FUNCTION FB_HEXSTR_TO_DINT																			// Converts a STRING hex array to DINT.
VAR_INPUT
	in						: STRING;																// The input string.
END_VAR
VAR_OUTPUT
	out						: DINT;																	// The output value.
	bError					: BOOL;																	// Had any error occured.
END_VAR
VAR
	sSum					: STRING;
	pVal					: PVOID;
END_VAR

// Converts a STRING hex array to DINT.
IF LEN(in) = 8 THEN
	sSum := CONCAT('16#', in);
	pVal := STRING_TO_PVOID(sSum);
	MEMCPY(ADR(out),
		ADR(pVal),
		4);
ELSE
	out := 0;
	bError := TRUE;
END_IF

END_FUNCTION

(* stored: Version 1.1.0.1, ProductVersion 3.1.4024.3
   POU FB_HEXSTR_TO_DINT: Id {df350655-9620-44a4-863d-d1cd4cd5df8c}, SpecialFunc None *)
